LIN {X 0,Y 116.552,Z 530.885,A -85,B 0,C 180,E1 -31515.249,E2 -31515.249} C_VEL
LIN {X 0,Y 105.346,Z 542.658,A -85,B 0,C 180,E1 -31515.432,E2 -31515.432} C_VEL
LIN {X 0,Y 93.073,Z 553.615,A -85,B 0,C 180,E1 -31515.684,E2 -31515.684} C_VEL
LIN {X 0,Y 80.4,Z 563.272,A -85,B 0,C 180,E1 -31515.939,E2 -31515.939} C_VEL
LIN {X 0,Y 65.877,Z 572.641,A -85,B 0,C 180,E1 -31516.224,E2 -31516.224} C_VEL
LIN {X 0,Y 51.34,Z 580.447,A -85,B 0,C 180,E1 -31516.611,E2 -31516.611} C_VEL
LIN {X 0,Y 36.719,Z 586.842,A -85,B 0,C 180,E1 -31516.856,E2 -31516.856} C_VEL
LIN {X 0,Y 21.968,Z 591.98,A -85,B 0,C 180,E1 -31516.291,E2 -31516.291} C_VEL
LIN {X 0,Y 14.491,Z 594.143,A -85,B 0,C 180,E1 -31514.042,E2 -31514.042} C_VEL
LIN {X 0,Y 14.431,Z 594.165,A -85,B 0,C 180,E1 -31513.05,E2 -31513.05} C_VEL
LIN {X 0,Y 28.679,Z 589.854,A -85,B 0,C 180,E1 -31511.393,E2 -31511.393} C_VEL
LIN {X 0,Y 43.003,Z 584.35,A -85,B 0,C 180,E1 -31511.298,E2 -31511.298} C_VEL
LIN {X 0,Y 57.366,Z 577.469,A -85,B 0,C 180,E1 -31511.445,E2 -31511.445} C_VEL
LIN {X 0,Y 71.738,Z 569.172,A -85,B 0,C 180,E1 -31511.565,E2 -31511.565} C_VEL
LIN {X 0,Y 84.313,Z 560.615,A -85,B 0,C 180,E1 -31511.637,E2 -31511.637} C_VEL
LIN {X 0,Y 96.926,Z 550.452,A -85,B 0,C 180,E1 -31511.796,E2 -31511.796} C_VEL
LIN {X 0,Y 109.514,Z 538.566,A -85,B 0,C 180,E1 -31511.856,E2 -31511.856} C_VEL
LIN {X 0,Y 121.185,Z 525.577,A -85,B 0,C 180,E1 -31511.86,E2 -31511.86} C_VEL
LIN {X 0,Y 131.015,Z 512.738,A -85,B 0,C 180,E1 -31511.905,E2 -31511.905} C_VEL
LIN {X 0,Y 140.052,Z 498.802,A -85,B 0,C 180,E1 -31511.892,E2 -31511.892} C_VEL
LIN {X 0,Y 148.15,Z 483.743,A -85,B 0,C 180,E1 -31511.925,E2 -31511.925} C_VEL
LIN {X 0,Y 154.883,Z 468.458,A -85,B 0,C 180,E1 -31511.924,E2 -31511.924} C_VEL
LIN {X 0,Y 160.577,Z 452.163,A -85,B 0,C 180,E1 -31511.914,E2 -31511.914} C_VEL
LIN {X 0,Y 164.925,Z 435.557,A -85,B 0,C 180,E1 -31511.862,E2 -31511.862} C_VEL
LIN {X 0,Y 166.898,Z 425.207,A -85,B 0,C 180,E1 -31511.993,E2 -31511.993} C_VEL
LIN {X 0,Y 166.84,Z 425.5,A -85,B 0,C 180,E1 -31514.173,E2 -31514.173} C_VEL
LIN {X 0,Y 166.836,Z 425.561,A -85,B 0,C 180,E1 -31514.384,E2 -31514.384} C_VEL
LIN {X 0,Y 163.983,Z 439.54,A -85,B 0,C 180,E1 -31514.465,E2 -31514.465} C_VEL
LIN {X 0,Y 163.923,Z 440.027,A -85,B 0,C 180,E1 -31514.467,E2 -31514.467} C_VEL
LIN {X 0,Y 163.923,Z 600,A -85,B 0,C 180,E1 -31514.467,E2 -31514.467} C_VEL
LIN {X 0,Y 163.923,Z 600,A -85,B 0,C 180,E1 -31514.467,E2 -31514.467}

QRS_NEXT_CUT()

QRS_NEXT()
QRS_HOME()

END
